TYPE ERROR_RECORD :
STRUCT
	Timer       : STRING;
	Axis        : UDINT;
	ErrorID     : UDINT;
	ErrorTXT    : STRING;
	ErrorCNT    : UDINT:=0;
END_STRUCT
END_TYPE

(* stored: Version 1.1.0.1, ProductVersion 3.1.4018.5
   DUT ERROR_RECORD: Id {9781350a-f4e2-4e68-89fe-e034c0ef55be} *)
